// TIA Portal V16 export
// export: Created 2021-11-12T13:32:55.8225279Z, ExportSetting WithDefaults, DisplayName Totally Integrated Automation Portal, DisplayVersion V16 Update 3, DisplayName TIA Portal Version Control Interface, DisplayVersion V16 Update 2, DisplayName TIA Portal Openness, DisplayVersion V16 Update 3, DisplayName SINAMICS Startdrive Advanced, DisplayVersion V16 Update 5, DisplayName SINAMICS Startdrive G130, G150, S120, S150, SINAMICS MV, S210, DisplayVersion V16 Update 5, DisplayName SINAMICS Startdrive G110M, G120, G120C, G120D, G120P, G115D, DisplayVersion V16 Update 5, DisplayName STEP 7 Professional, DisplayVersion V16 Update 3, DisplayName STEP 7 Safety, DisplayVersion V16, DisplayName WinCC UA Professional, DisplayVersion V16 Update 3
FUNCTION_BLOCK "IM_300+UH11-KF10"   // FB64, LAD
TITLE = Inputs reading
{ S7_Optimized_Access := 'TRUE' }
VERSION : 0.1
// MICE Wood interface block
// stored: AutoNumber true, IsIECCheckEnabled false, IsRetainMemResEnabled false, MemoryReserve 100, SetENOAutomatically false, UDAEnableTagReadback false
   VAR
      KF11_Ix0 { S7_SetPoint := 'True'} : "STD_CH_DI";
      KF11_Ix1 { S7_SetPoint := 'True'} : "STD_CH_DI";
      KF11_Ix2 { S7_SetPoint := 'True'} : "STD_CH_DI";
      KF11_Ix3 { S7_SetPoint := 'True'} : "STD_CH_DI";
      KF11_Ix4 { S7_SetPoint := 'True'} : "STD_CH_DI";
      KF11_Ix5 { S7_SetPoint := 'True'} : "STD_CH_DI";
      KF11_Ix6 { S7_SetPoint := 'True'} : "STD_CH_DI";
      KF11_Ix7 { S7_SetPoint := 'True'} : "STD_CH_DI";
      KF11_Ix8 { S7_SetPoint := 'True'} : "STD_CH_DI";
      KF11_Ix9 { S7_SetPoint := 'True'} : "STD_CH_DI";
      KF11_Ix10 { S7_SetPoint := 'True'} : "STD_CH_DI";
      KF11_Ix11 { S7_SetPoint := 'True'} : "STD_CH_DI";
      KF11_Ix12 { S7_SetPoint := 'True'} : "STD_CH_DI";
      KF11_Ix13 { S7_SetPoint := 'True'} : "STD_CH_DI";
      KF11_Ix14 { S7_SetPoint := 'True'} : "STD_CH_DI";
      KF11_Ix15 { S7_SetPoint := 'True'} : "STD_CH_DI";
      KF12_Ix0 { S7_SetPoint := 'True'} : "STD_CH_DI";
      KF12_Ix1 { S7_SetPoint := 'True'} : "STD_CH_DI";
      KF12_Ix2 { S7_SetPoint := 'True'} : "STD_CH_DI";
      KF12_Ix3 { S7_SetPoint := 'True'} : "STD_CH_DI";
      KF12_Ix4 { S7_SetPoint := 'True'} : "STD_CH_DI";
      KF12_Ix5 { S7_SetPoint := 'True'} : "STD_CH_DI";
      KF12_Ix6 { S7_SetPoint := 'True'} : "STD_CH_DI";
      KF12_Ix7 { S7_SetPoint := 'True'} : "STD_CH_DI";
      KF13_Ix0 { S7_SetPoint := 'True'} : "STD_CH_DI";
      KF13_Ix1 { S7_SetPoint := 'True'} : "STD_CH_DI";
      KF13_Ix2 { S7_SetPoint := 'True'} : "STD_CH_DI";
      KF13_Ix3 { S7_SetPoint := 'True'} : "STD_CH_DI";
      KF13_Ix4 { S7_SetPoint := 'True'} : "STD_CH_DI";
      KF13_Ix5 { S7_SetPoint := 'True'} : "STD_CH_DI";
      KF13_Ix6 { S7_SetPoint := 'True'} : "STD_CH_DI";
      KF13_Ix7 { S7_SetPoint := 'True'} : "STD_CH_DI";
      KF13_Ix8 { S7_SetPoint := 'True'} : "STD_CH_DI";
      KF13_Ix9 { S7_SetPoint := 'True'} : "STD_CH_DI";
      KF13_Ix10 { S7_SetPoint := 'True'} : "STD_CH_DI";
      KF13_Ix11 { S7_SetPoint := 'True'} : "STD_CH_DI";
      KF13_Ix12 { S7_SetPoint := 'True'} : "STD_CH_DI";
      KF13_Ix13 { S7_SetPoint := 'True'} : "STD_CH_DI";
      KF13_Ix14 { S7_SetPoint := 'True'} : "STD_CH_DI";
      KF13_Ix15 { S7_SetPoint := 'True'} : "STD_CH_DI";
      KF14_Ix0 { S7_SetPoint := 'True'} : "STD_CH_DI";
      KF14_Ix1 { S7_SetPoint := 'True'} : "STD_CH_DI";
      KF14_Ix2 { S7_SetPoint := 'True'} : "STD_CH_DI";
      KF14_Ix3 { S7_SetPoint := 'True'} : "STD_CH_DI";
      KF14_Ix4 { S7_SetPoint := 'True'} : "STD_CH_DI";
      KF14_Ix5 { S7_SetPoint := 'True'} : "STD_CH_DI";
      KF14_Ix6 { S7_SetPoint := 'True'} : "STD_CH_DI";
      KF14_Ix7 { S7_SetPoint := 'True'} : "STD_CH_DI";
      KF14_Ix8 { S7_SetPoint := 'True'} : "STD_CH_DI";
      KF14_Ix9 { S7_SetPoint := 'True'} : "STD_CH_DI";
      KF14_Ix10 { S7_SetPoint := 'True'} : "STD_CH_DI";
      KF14_Ix11 { S7_SetPoint := 'True'} : "STD_CH_DI";
      KF14_Ix12 { S7_SetPoint := 'True'} : "STD_CH_DI";
      KF14_Ix13 { S7_SetPoint := 'True'} : "STD_CH_DI";
      KF14_Ix14 { S7_SetPoint := 'True'} : "STD_CH_DI";
      KF14_Ix15 { S7_SetPoint := 'True'} : "STD_CH_DI";
      KF15_Ix0 { S7_SetPoint := 'True'} : "STD_CH_DI";
      KF15_Ix1 { S7_SetPoint := 'True'} : "STD_CH_DI";
      KF15_Ix2 { S7_SetPoint := 'True'} : "STD_CH_DI";
      KF15_Ix3 { S7_SetPoint := 'True'} : "STD_CH_DI";
      KF15_Ix4 { S7_SetPoint := 'True'} : "STD_CH_DI";
      KF15_Ix5 { S7_SetPoint := 'True'} : "STD_CH_DI";
      KF15_Ix6 { S7_SetPoint := 'True'} : "STD_CH_DI";
      KF15_Ix7 { S7_SetPoint := 'True'} : "STD_CH_DI";
      KF15_Ix8 { S7_SetPoint := 'True'} : "STD_CH_DI";
      KF15_Ix9 { S7_SetPoint := 'True'} : "STD_CH_DI";
      KF15_Ix10 { S7_SetPoint := 'True'} : "STD_CH_DI";
      KF15_Ix11 { S7_SetPoint := 'True'} : "STD_CH_DI";
      KF15_Ix12 { S7_SetPoint := 'True'} : "STD_CH_DI";
      KF15_Ix13 { S7_SetPoint := 'True'} : "STD_CH_DI";
      KF15_Ix14 { S7_SetPoint := 'True'} : "STD_CH_DI";
      KF15_Ix15 { S7_SetPoint := 'True'} : "STD_CH_DI";
      KF61_AI0 { S7_SetPoint := 'True'} : "STD_CH_AI";
      KF61_AI1 { S7_SetPoint := 'True'} : "STD_CH_AI";
      KF61_AI2 { S7_SetPoint := 'True'} : "STD_CH_AI";
      KF61_AI3 { S7_SetPoint := 'True'} : "STD_CH_AI";
   END_VAR
   VAR_TEMP   // added for the SCL form of the ladder/FBD networks
      _w1 : Bool;
      _w2 : Bool;
      _w3 : Bool;
      _w4 : Bool;
      _w5 : Bool;
      _w6 : Bool;
      _w7 : Bool;
      _w8 : Bool;
   END_VAR
BEGIN

REGION Network 1: Module position -KF11
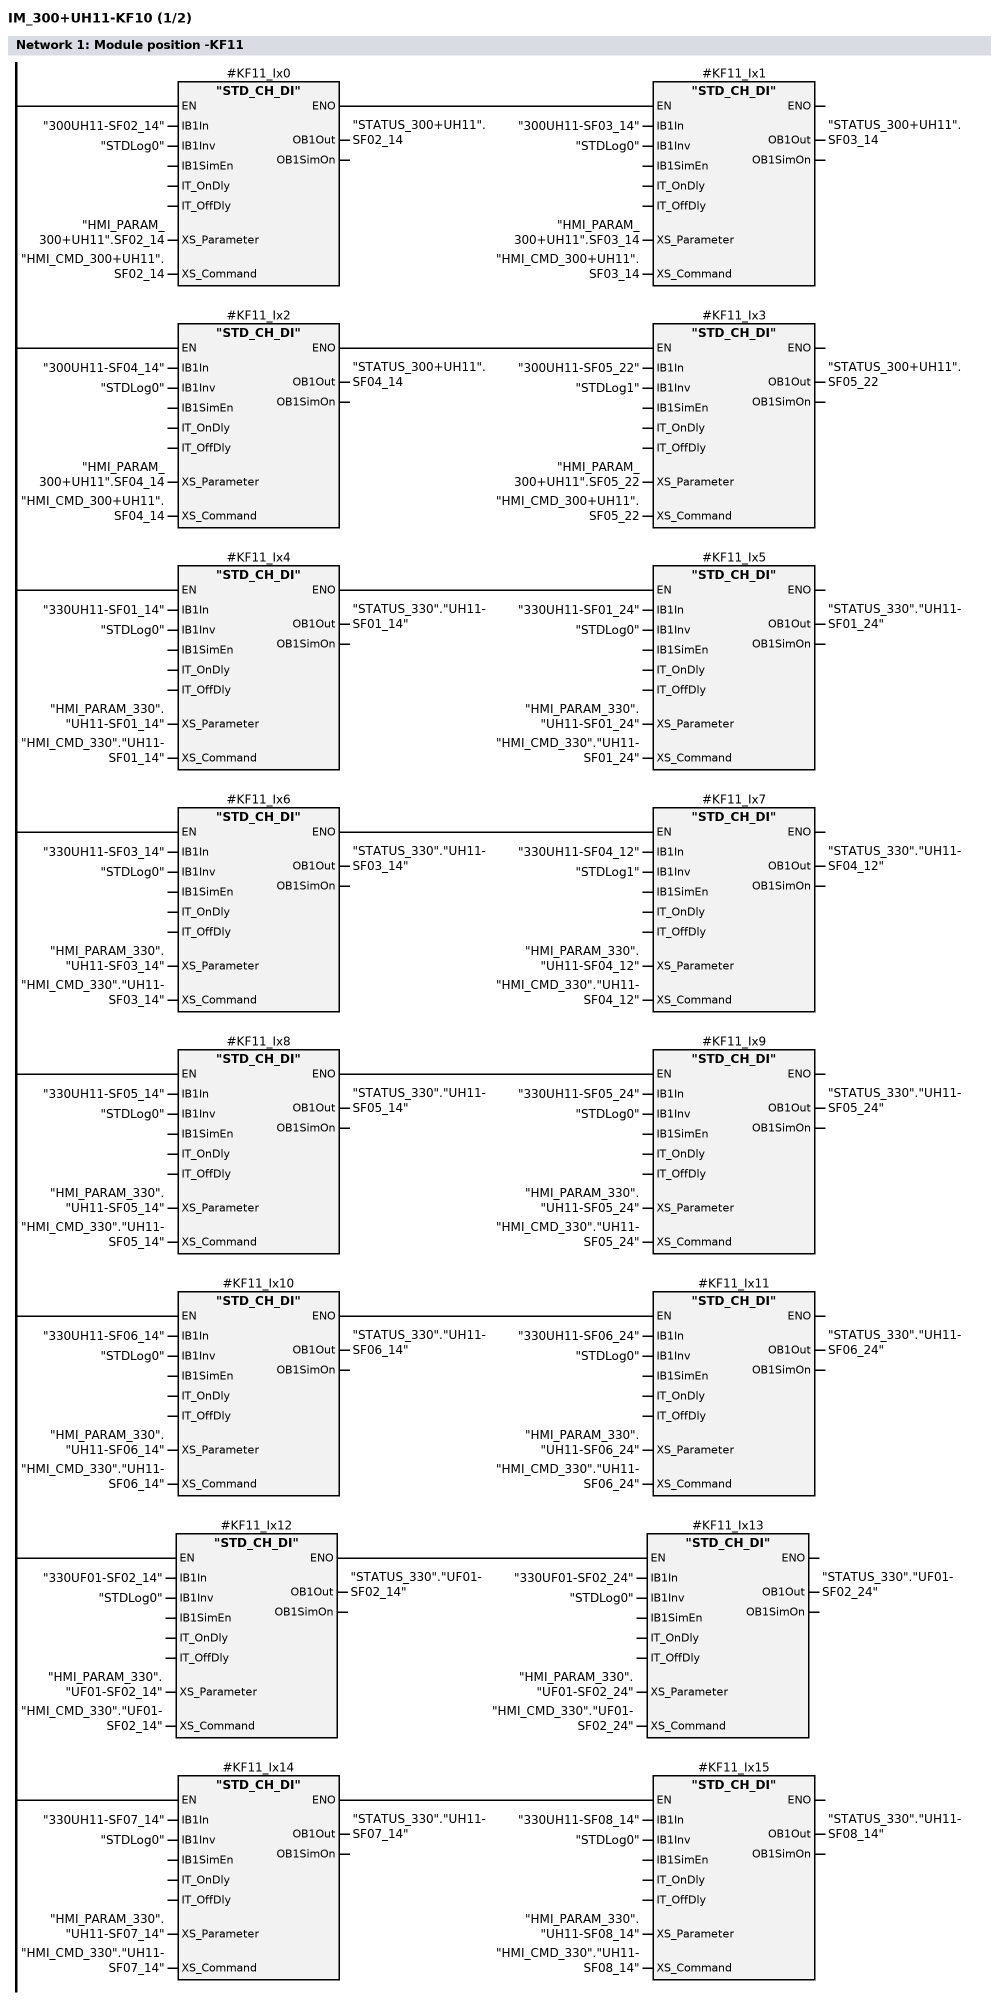
   RUNG wire#powerrail
      #KF11_Ix0(IB1In := "300UH11-SF02_14", IB1Inv := "STDLog0", IB1SimEn :=, IT_OnDly :=, IT_OffDly :=, XS_Parameter := "HMI_PARAM_300+UH11".SF02_14, XS_Command := "HMI_CMD_300+UH11".SF02_14, OB1Out => "STATUS_300+UH11".SF02_14, OB1SimOn =>)
      #KF11_Ix1(IB1In := "300UH11-SF03_14", IB1Inv := "STDLog0", IB1SimEn :=, IT_OnDly :=, IT_OffDly :=, XS_Parameter := "HMI_PARAM_300+UH11".SF03_14, XS_Command := "HMI_CMD_300+UH11".SF03_14, OB1Out => "STATUS_300+UH11".SF03_14, OB1SimOn =>)
   END_RUNG
   RUNG wire#powerrail
      #KF11_Ix2(IB1In := "300UH11-SF04_14", IB1Inv := "STDLog0", IB1SimEn :=, IT_OnDly :=, IT_OffDly :=, XS_Parameter := "HMI_PARAM_300+UH11".SF04_14, XS_Command := "HMI_CMD_300+UH11".SF04_14, OB1Out => "STATUS_300+UH11".SF04_14, OB1SimOn =>)
      #KF11_Ix3(IB1In := "300UH11-SF05_22", IB1Inv := "STDLog1", IB1SimEn :=, IT_OnDly :=, IT_OffDly :=, XS_Parameter := "HMI_PARAM_300+UH11".SF05_22, XS_Command := "HMI_CMD_300+UH11".SF05_22, OB1Out => "STATUS_300+UH11".SF05_22, OB1SimOn =>)
   END_RUNG
   RUNG wire#powerrail
      #KF11_Ix4(IB1In := "330UH11-SF01_14", IB1Inv := "STDLog0", IB1SimEn :=, IT_OnDly :=, IT_OffDly :=, XS_Parameter := "HMI_PARAM_330"."UH11-SF01_14", XS_Command := "HMI_CMD_330"."UH11-SF01_14", OB1Out => "STATUS_330"."UH11-SF01_14", OB1SimOn =>)
      #KF11_Ix5(IB1In := "330UH11-SF01_24", IB1Inv := "STDLog0", IB1SimEn :=, IT_OnDly :=, IT_OffDly :=, XS_Parameter := "HMI_PARAM_330"."UH11-SF01_24", XS_Command := "HMI_CMD_330"."UH11-SF01_24", OB1Out => "STATUS_330"."UH11-SF01_24", OB1SimOn =>)
   END_RUNG
   RUNG wire#powerrail
      #KF11_Ix6(IB1In := "330UH11-SF03_14", IB1Inv := "STDLog0", IB1SimEn :=, IT_OnDly :=, IT_OffDly :=, XS_Parameter := "HMI_PARAM_330"."UH11-SF03_14", XS_Command := "HMI_CMD_330"."UH11-SF03_14", OB1Out => "STATUS_330"."UH11-SF03_14", OB1SimOn =>)
      #KF11_Ix7(IB1In := "330UH11-SF04_12", IB1Inv := "STDLog1", IB1SimEn :=, IT_OnDly :=, IT_OffDly :=, XS_Parameter := "HMI_PARAM_330"."UH11-SF04_12", XS_Command := "HMI_CMD_330"."UH11-SF04_12", OB1Out => "STATUS_330"."UH11-SF04_12", OB1SimOn =>)
   END_RUNG
   RUNG wire#powerrail
      #KF11_Ix8(IB1In := "330UH11-SF05_14", IB1Inv := "STDLog0", IB1SimEn :=, IT_OnDly :=, IT_OffDly :=, XS_Parameter := "HMI_PARAM_330"."UH11-SF05_14", XS_Command := "HMI_CMD_330"."UH11-SF05_14", OB1Out => "STATUS_330"."UH11-SF05_14", OB1SimOn =>)
      #KF11_Ix9(IB1In := "330UH11-SF05_24", IB1Inv := "STDLog0", IB1SimEn :=, IT_OnDly :=, IT_OffDly :=, XS_Parameter := "HMI_PARAM_330"."UH11-SF05_24", XS_Command := "HMI_CMD_330"."UH11-SF05_24", OB1Out => "STATUS_330"."UH11-SF05_24", OB1SimOn =>)
   END_RUNG
   RUNG wire#powerrail
      #KF11_Ix10(IB1In := "330UH11-SF06_14", IB1Inv := "STDLog0", IB1SimEn :=, IT_OnDly :=, IT_OffDly :=, XS_Parameter := "HMI_PARAM_330"."UH11-SF06_14", XS_Command := "HMI_CMD_330"."UH11-SF06_14", OB1Out => "STATUS_330"."UH11-SF06_14", OB1SimOn =>)
      #KF11_Ix11(IB1In := "330UH11-SF06_24", IB1Inv := "STDLog0", IB1SimEn :=, IT_OnDly :=, IT_OffDly :=, XS_Parameter := "HMI_PARAM_330"."UH11-SF06_24", XS_Command := "HMI_CMD_330"."UH11-SF06_24", OB1Out => "STATUS_330"."UH11-SF06_24", OB1SimOn =>)
   END_RUNG
   RUNG wire#powerrail
      #KF11_Ix12(IB1In := "330UF01-SF02_14", IB1Inv := "STDLog0", IB1SimEn :=, IT_OnDly :=, IT_OffDly :=, XS_Parameter := "HMI_PARAM_330"."UF01-SF02_14", XS_Command := "HMI_CMD_330"."UF01-SF02_14", OB1Out => "STATUS_330"."UF01-SF02_14", OB1SimOn =>)
      #KF11_Ix13(IB1In := "330UF01-SF02_24", IB1Inv := "STDLog0", IB1SimEn :=, IT_OnDly :=, IT_OffDly :=, XS_Parameter := "HMI_PARAM_330"."UF01-SF02_24", XS_Command := "HMI_CMD_330"."UF01-SF02_24", OB1Out => "STATUS_330"."UF01-SF02_24", OB1SimOn =>)
   END_RUNG
   RUNG wire#powerrail
      #KF11_Ix14(IB1In := "330UH11-SF07_14", IB1Inv := "STDLog0", IB1SimEn :=, IT_OnDly :=, IT_OffDly :=, XS_Parameter := "HMI_PARAM_330"."UH11-SF07_14", XS_Command := "HMI_CMD_330"."UH11-SF07_14", OB1Out => "STATUS_330"."UH11-SF07_14", OB1SimOn =>)
      #KF11_Ix15(IB1In := "330UH11-SF08_14", IB1Inv := "STDLog0", IB1SimEn :=, IT_OnDly :=, IT_OffDly :=, XS_Parameter := "HMI_PARAM_330"."UH11-SF08_14", XS_Command := "HMI_CMD_330"."UH11-SF08_14", OB1Out => "STATUS_330"."UH11-SF08_14", OB1SimOn =>)
   END_RUNG
   // the same network as SCL:
   #KF11_Ix0(IB1In := "300UH11-SF02_14",   // "STD_CH_DI"
             IB1Inv := "STDLog0",
             XS_Parameter := "HMI_PARAM_300+UH11".SF02_14,
             XS_Command := "HMI_CMD_300+UH11".SF02_14,
             OB1Out => "STATUS_300+UH11".SF02_14,
             ENO => #_w1);
   IF #_w1 THEN
       #KF11_Ix1(IB1In := "300UH11-SF03_14",   // "STD_CH_DI"
                 IB1Inv := "STDLog0",
                 XS_Parameter := "HMI_PARAM_300+UH11".SF03_14,
                 XS_Command := "HMI_CMD_300+UH11".SF03_14,
                 OB1Out => "STATUS_300+UH11".SF03_14);
   END_IF;
   #KF11_Ix2(IB1In := "300UH11-SF04_14",   // "STD_CH_DI"
             IB1Inv := "STDLog0",
             XS_Parameter := "HMI_PARAM_300+UH11".SF04_14,
             XS_Command := "HMI_CMD_300+UH11".SF04_14,
             OB1Out => "STATUS_300+UH11".SF04_14,
             ENO => #_w2);
   IF #_w2 THEN
       #KF11_Ix3(IB1In := "300UH11-SF05_22",   // "STD_CH_DI"
                 IB1Inv := "STDLog1",
                 XS_Parameter := "HMI_PARAM_300+UH11".SF05_22,
                 XS_Command := "HMI_CMD_300+UH11".SF05_22,
                 OB1Out => "STATUS_300+UH11".SF05_22);
   END_IF;
   #KF11_Ix4(IB1In := "330UH11-SF01_14",   // "STD_CH_DI"
             IB1Inv := "STDLog0",
             XS_Parameter := "HMI_PARAM_330"."UH11-SF01_14",
             XS_Command := "HMI_CMD_330"."UH11-SF01_14",
             OB1Out => "STATUS_330"."UH11-SF01_14",
             ENO => #_w3);
   IF #_w3 THEN
       #KF11_Ix5(IB1In := "330UH11-SF01_24",   // "STD_CH_DI"
                 IB1Inv := "STDLog0",
                 XS_Parameter := "HMI_PARAM_330"."UH11-SF01_24",
                 XS_Command := "HMI_CMD_330"."UH11-SF01_24",
                 OB1Out => "STATUS_330"."UH11-SF01_24");
   END_IF;
   #KF11_Ix6(IB1In := "330UH11-SF03_14",   // "STD_CH_DI"
             IB1Inv := "STDLog0",
             XS_Parameter := "HMI_PARAM_330"."UH11-SF03_14",
             XS_Command := "HMI_CMD_330"."UH11-SF03_14",
             OB1Out => "STATUS_330"."UH11-SF03_14",
             ENO => #_w4);
   IF #_w4 THEN
       #KF11_Ix7(IB1In := "330UH11-SF04_12",   // "STD_CH_DI"
                 IB1Inv := "STDLog1",
                 XS_Parameter := "HMI_PARAM_330"."UH11-SF04_12",
                 XS_Command := "HMI_CMD_330"."UH11-SF04_12",
                 OB1Out => "STATUS_330"."UH11-SF04_12");
   END_IF;
   #KF11_Ix8(IB1In := "330UH11-SF05_14",   // "STD_CH_DI"
             IB1Inv := "STDLog0",
             XS_Parameter := "HMI_PARAM_330"."UH11-SF05_14",
             XS_Command := "HMI_CMD_330"."UH11-SF05_14",
             OB1Out => "STATUS_330"."UH11-SF05_14",
             ENO => #_w5);
   IF #_w5 THEN
       #KF11_Ix9(IB1In := "330UH11-SF05_24",   // "STD_CH_DI"
                 IB1Inv := "STDLog0",
                 XS_Parameter := "HMI_PARAM_330"."UH11-SF05_24",
                 XS_Command := "HMI_CMD_330"."UH11-SF05_24",
                 OB1Out => "STATUS_330"."UH11-SF05_24");
   END_IF;
   #KF11_Ix10(IB1In := "330UH11-SF06_14",   // "STD_CH_DI"
              IB1Inv := "STDLog0",
              XS_Parameter := "HMI_PARAM_330"."UH11-SF06_14",
              XS_Command := "HMI_CMD_330"."UH11-SF06_14",
              OB1Out => "STATUS_330"."UH11-SF06_14",
              ENO => #_w6);
   IF #_w6 THEN
       #KF11_Ix11(IB1In := "330UH11-SF06_24",   // "STD_CH_DI"
                  IB1Inv := "STDLog0",
                  XS_Parameter := "HMI_PARAM_330"."UH11-SF06_24",
                  XS_Command := "HMI_CMD_330"."UH11-SF06_24",
                  OB1Out => "STATUS_330"."UH11-SF06_24");
   END_IF;
   #KF11_Ix12(IB1In := "330UF01-SF02_14",   // "STD_CH_DI"
              IB1Inv := "STDLog0",
              XS_Parameter := "HMI_PARAM_330"."UF01-SF02_14",
              XS_Command := "HMI_CMD_330"."UF01-SF02_14",
              OB1Out => "STATUS_330"."UF01-SF02_14",
              ENO => #_w7);
   IF #_w7 THEN
       #KF11_Ix13(IB1In := "330UF01-SF02_24",   // "STD_CH_DI"
                  IB1Inv := "STDLog0",
                  XS_Parameter := "HMI_PARAM_330"."UF01-SF02_24",
                  XS_Command := "HMI_CMD_330"."UF01-SF02_24",
                  OB1Out => "STATUS_330"."UF01-SF02_24");
   END_IF;
   #KF11_Ix14(IB1In := "330UH11-SF07_14",   // "STD_CH_DI"
              IB1Inv := "STDLog0",
              XS_Parameter := "HMI_PARAM_330"."UH11-SF07_14",
              XS_Command := "HMI_CMD_330"."UH11-SF07_14",
              OB1Out => "STATUS_330"."UH11-SF07_14",
              ENO => #_w8);
   IF #_w8 THEN
       #KF11_Ix15(IB1In := "330UH11-SF08_14",   // "STD_CH_DI"
                  IB1Inv := "STDLog0",
                  XS_Parameter := "HMI_PARAM_330"."UH11-SF08_14",
                  XS_Command := "HMI_CMD_330"."UH11-SF08_14",
                  OB1Out => "STATUS_330"."UH11-SF08_14");
   END_IF;
END_REGION

REGION Network 2: Module position -KF12
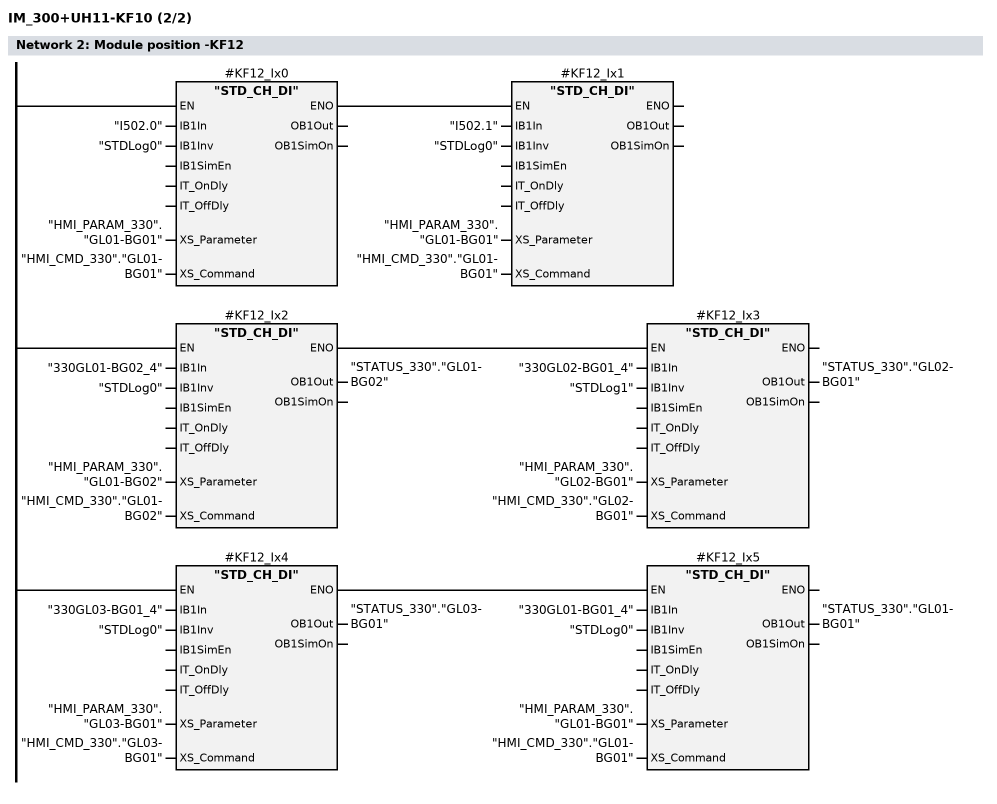
   RUNG wire#powerrail
      #KF12_Ix0(IB1In := "I502.0", IB1Inv := "STDLog0", IB1SimEn :=, IT_OnDly :=, IT_OffDly :=, XS_Parameter := "HMI_PARAM_330"."GL01-BG01", XS_Command := "HMI_CMD_330"."GL01-BG01", OB1Out =>, OB1SimOn =>)
      #KF12_Ix1(IB1In := "I502.1", IB1Inv := "STDLog0", IB1SimEn :=, IT_OnDly :=, IT_OffDly :=, XS_Parameter := "HMI_PARAM_330"."GL01-BG01", XS_Command := "HMI_CMD_330"."GL01-BG01", OB1Out =>, OB1SimOn =>)
   END_RUNG
   RUNG wire#powerrail
      #KF12_Ix2(IB1In := "330GL01-BG02_4", IB1Inv := "STDLog0", IB1SimEn :=, IT_OnDly :=, IT_OffDly :=, XS_Parameter := "HMI_PARAM_330"."GL01-BG02", XS_Command := "HMI_CMD_330"."GL01-BG02", OB1Out => "STATUS_330"."GL01-BG02", OB1SimOn =>)
      #KF12_Ix3(IB1In := "330GL02-BG01_4", IB1Inv := "STDLog1", IB1SimEn :=, IT_OnDly :=, IT_OffDly :=, XS_Parameter := "HMI_PARAM_330"."GL02-BG01", XS_Command := "HMI_CMD_330"."GL02-BG01", OB1Out => "STATUS_330"."GL02-BG01", OB1SimOn =>)
   END_RUNG
   RUNG wire#powerrail
      #KF12_Ix4(IB1In := "330GL03-BG01_4", IB1Inv := "STDLog0", IB1SimEn :=, IT_OnDly :=, IT_OffDly :=, XS_Parameter := "HMI_PARAM_330"."GL03-BG01", XS_Command := "HMI_CMD_330"."GL03-BG01", OB1Out => "STATUS_330"."GL03-BG01", OB1SimOn =>)
      #KF12_Ix5(IB1In := "330GL01-BG01_4", IB1Inv := "STDLog0", IB1SimEn :=, IT_OnDly :=, IT_OffDly :=, XS_Parameter := "HMI_PARAM_330"."GL01-BG01", XS_Command := "HMI_CMD_330"."GL01-BG01", OB1Out => "STATUS_330"."GL01-BG01", OB1SimOn =>)
   END_RUNG
   // the same network as SCL:
   #KF12_Ix0(IB1In := "I502.0",   // "STD_CH_DI"
             IB1Inv := "STDLog0",
             XS_Parameter := "HMI_PARAM_330"."GL01-BG01",
             XS_Command := "HMI_CMD_330"."GL01-BG01",
             ENO => #_w1);
   IF #_w1 THEN
       #KF12_Ix1(IB1In := "I502.1",   // "STD_CH_DI"
                 IB1Inv := "STDLog0",
                 XS_Parameter := "HMI_PARAM_330"."GL01-BG01",
                 XS_Command := "HMI_CMD_330"."GL01-BG01");
   END_IF;
   #KF12_Ix2(IB1In := "330GL01-BG02_4",   // "STD_CH_DI"
             IB1Inv := "STDLog0",
             XS_Parameter := "HMI_PARAM_330"."GL01-BG02",
             XS_Command := "HMI_CMD_330"."GL01-BG02",
             OB1Out => "STATUS_330"."GL01-BG02",
             ENO => #_w2);
   IF #_w2 THEN
       #KF12_Ix3(IB1In := "330GL02-BG01_4",   // "STD_CH_DI"
                 IB1Inv := "STDLog1",
                 XS_Parameter := "HMI_PARAM_330"."GL02-BG01",
                 XS_Command := "HMI_CMD_330"."GL02-BG01",
                 OB1Out => "STATUS_330"."GL02-BG01");
   END_IF;
   #KF12_Ix4(IB1In := "330GL03-BG01_4",   // "STD_CH_DI"
             IB1Inv := "STDLog0",
             XS_Parameter := "HMI_PARAM_330"."GL03-BG01",
             XS_Command := "HMI_CMD_330"."GL03-BG01",
             OB1Out => "STATUS_330"."GL03-BG01",
             ENO => #_w3);
   IF #_w3 THEN
       #KF12_Ix5(IB1In := "330GL01-BG01_4",   // "STD_CH_DI"
                 IB1Inv := "STDLog0",
                 XS_Parameter := "HMI_PARAM_330"."GL01-BG01",
                 XS_Command := "HMI_CMD_330"."GL01-BG01",
                 OB1Out => "STATUS_330"."GL01-BG01");
   END_IF;
END_REGION
END_FUNCTION_BLOCK
